Yaskawa INFORM job: R1_W14,16(0,0)OK-KM.JBI

/JOB
//NAME R1_W14,16(0,0)OK-KM
///FOLDERNAME KRIS-SCIANA
//POS
///NPOS 101,101,0,6,0,0
///TOOL 0
///POSTYPE PULSE
///PULSE
C00000=77640,24989,-13034,1442,74650,-81979
C00001=222133,14236,-6582,35909,75412,-22741
C00002=224151,18213,-1142,35502,73514,-22529
C00003=224936,19873,1121,35352,72748,-22454
C00004=225158,22602,3700,35316,72503,-22444
C00005=224936,19873,1121,35352,72748,-22454
C00006=225492,20065,2012,35260,72151,-22417
C00007=225492,20150,3698,35437,71333,-22690
C00008=225492,20065,2012,35260,72151,-22417
C00009=225905,19824,2070,35161,71851,-22342
C00010=226863,19321,1598,34859,71490,-22055
C00011=225905,19824,2070,35161,71851,-22342
C00012=225128,18122,-233,35305,72616,-22417
C00013=223128,14040,-5766,35700,74509,-22627
C00014=220661,2218,-15559,48375,67876,-23710
C00015=223949,9044,-9659,47271,66070,-22948
C00016=224087,10523,-8349,47237,65966,-22927
C00017=224042,10033,-8784,47248,66001,-22933
C00018=224042,10033,-8784,47248,66001,-22933
C00019=224745,9640,-9133,46989,65646,-22751
C00020=223995,9217,-9507,47256,66043,-22935
C00021=219810,-7663,-21002,65356,59757,-26400
C00022=222255,-3125,-17635,64445,58296,-25854
C00023=223197,-1261,-16218,64086,57730,-25645
C00024=223480,1501,-13911,63991,57548,-25594
C00025=223197,-1261,-16218,64086,57730,-25645
C00026=223908,-1254,-16349,63799,57315,-25476
C00027=225105,-1875,-16864,63387,56549,-25256
C00028=223908,-1254,-16349,63799,57315,-25476
C00029=223463,-1317,-18857,63116,58306,-24835
C00030=223463,-1302,-19472,62908,58490,-24651
C00031=223424,-1704,-17925,63552,57967,-25210
C00032=222481,-3577,-19346,63923,58526,-25421
C00033=220036,-8144,-22725,64866,59971,-25975
C00034=226102,-30423,-43926,14586,59978,3306
C00035=229259,38452,3699,-28321,84051,11178
C00036=227866,42540,10325,-28019,81848,11201
C00037=226976,47240,16142,-27837,80525,11190
C00038=226976,47162,16651,-27859,80211,11267
C00039=226976,47240,16142,-27837,80525,11190
C00040=223490,38048,5548,-21341,76491,4888
C00041=223597,39362,6909,-21393,76366,4949
C00042=225154,40482,8624,-23914,78071,7653
C00043=226382,33405,5149,-28983,73314,10641
C00044=225848,33713,5458,-28793,73102,10489
C00045=226800,33173,4915,-29132,73476,10760
C00046=227343,31188,2133,-29239,74267,10763
C00047=228749,26406,-4564,-29549,76202,10795
C00048=232070,-21849,-33765,-61090,62787,20907
C00049=228897,-69525,-52932,-81421,40129,27644
C00050=227458,-1039,11305,-103194,37608,33319
C00051=224958,9874,17770,-101661,35535,32336
C00052=224188,13683,20614,-101562,34950,32247
C00053=224309,15055,21867,-101627,35049,32289
C00054=224188,13683,20614,-101562,34950,32247
C00055=228943,22603,28948,-98890,46973,31456
C00056=228371,22871,29203,-99004,46566,31500
C00057=230119,20169,17224,-83081,48510,27787
C00058=230119,19939,16315,-82693,48579,27522
C00059=230119,20412,18152,-83475,48444,28057
C00060=230834,18316,16575,-83629,48946,28167
C00061=237272,-16480,-7416,-86396,53244,30318
C00062=226102,-30423,-43926,14586,59978,18513
C00063=216741,-24945,-44490,70900,55443,-67548
C00064=233770,-38242,-44235,89025,19285,-70455
C00065=232263,-12981,-20271,101799,31607,-56551
C00066=225008,-3810,-25351,68302,49674,-66777
C00067=224928,-2342,-24150,68324,49732,-66782
C00068=232472,-143,20091,126873,38436,-70149
C00069=232295,-11422,-4289,83587,31547,-48271
C00070=235949,-23068,-3497,134153,23753,-86044
C00071=221775,-4145,-3632,80714,47909,-75071
C00072=221868,-5805,-11746,98440,47173,-76002
C00073=224762,-3456,-10718,97920,45016,-75779
C00074=212311,-14192,-18848,96672,72508,-34975
C00075=225062,-3438,-11050,97706,44778,-75655
C00076=224981,-1976,-9851,97692,44835,-75643
C00077=212303,2769,29618,102443,75165,-45073
C00078=223552,-52882,-25947,90849,39544,-36058
C00079=221750,-4780,-5976,79726,48150,-74402
C00080=222455,-35947,-31649,13557,42914,-27667
C00081=237520,-26297,-36521,-56184,44849,52997
C00082=227430,-8986,2777,-105996,27008,67297
C00083=226046,668,8189,-102778,26699,65688
C00084=225096,7310,14013,-103452,26054,65991
C00085=227562,6691,-16510,-46000,42357,47609
C00086=227319,5585,-17469,-45803,42251,47516
C00087=224970,42335,84441,-140073,39060,85063
C00088=224879,29476,62062,-121250,29359,73886
C00089=227160,29335,71248,-136736,39012,83614
C00090=229934,2939,2236,-61070,35416,56138
C00091=229942,357,-16619,-50330,41431,49996
C00092=230607,-744,-7505,-83554,33312,60975
C00093=228290,3572,-4729,-82188,31724,60324
C00094=227452,5680,-3434,-81484,31174,59986
C00095=228279,4951,-3893,-81869,31750,60157
C00096=228037,3832,-4852,-81778,31579,60118
C00097=227208,23451,46622,-116903,33779,78542
C00098=230396,11237,36356,-114852,35808,77806
C00099=237476,-68885,-64231,-58705,66532,55214
C00100=145215,-69093,-87212,-37312,66696,68321
BC00000=241198,366988,1031591
BC00001=398174,77442,788239
BC00002=398174,77442,788239
BC00003=398174,77442,788239
BC00004=398174,77442,788239
BC00005=398174,77442,788239
BC00006=398174,77442,788239
BC00007=398174,77442,788239
BC00008=398174,77442,788239
BC00009=398174,77442,788239
BC00010=398174,77442,788239
BC00011=398174,77442,788239
BC00012=398174,77442,788239
BC00013=398174,77442,788239
BC00014=398174,70944,901946
BC00015=398174,70944,901946
BC00016=398174,70944,901946
BC00017=398174,70944,901946
BC00018=398174,70944,901946
BC00019=398174,70944,901946
BC00020=398174,70944,901946
BC00021=398174,63251,1036573
BC00022=398174,63251,1036573
BC00023=398174,63251,1036573
BC00024=398174,63251,1036573
BC00025=398174,63251,1036573
BC00026=398174,63251,1036573
BC00027=398174,63251,1036573
BC00028=398174,63251,1036573
BC00029=398174,63251,1036573
BC00030=398174,63251,1036573
BC00031=398174,63251,1036573
BC00032=398174,63251,1036573
BC00033=398174,63251,1036573
BC00034=398174,59868,1073520
BC00035=398174,86212,734350
BC00036=398174,86212,734350
BC00037=398174,86212,734350
BC00038=398174,86212,734350
BC00039=398174,86212,734350
BC00040=398174,86212,734350
BC00041=398174,86212,734350
BC00042=398174,86212,734350
BC00043=398174,86212,734350
BC00044=398174,86212,734350
BC00045=398174,86212,734350
BC00046=398174,86212,734350
BC00047=398174,86212,734350
BC00048=398174,98499,866647
BC00049=398174,100680,959819
BC00050=398174,103382,1075175
BC00051=398174,103382,1075175
BC00052=398174,103382,1075175
BC00053=398174,103382,1075175
BC00054=398174,103382,1075175
BC00055=398174,103382,1075175
BC00056=398174,103382,1075175
BC00057=398174,103382,1075175
BC00058=398174,103382,1075175
BC00059=398174,103382,1075175
BC00060=398174,103382,1075175
BC00061=398174,103382,1075175
BC00062=395324,71612,1073520
BC00063=398174,59556,681470
BC00064=398173,59556,681467
BC00065=398172,59557,681466
BC00066=398174,59556,681470
BC00067=398174,59556,681470
BC00068=398172,59557,681466
BC00069=398172,59557,681466
BC00070=398173,59556,681467
BC00071=398174,59556,681470
BC00072=398174,59378,943465
BC00073=398174,59378,943465
BC00074=355798,67513,940049
BC00075=398174,59378,943465
BC00076=398174,59378,943465
BC00077=355868,67500,939621
BC00078=355790,67515,940051
BC00079=398174,59378,943465
BC00080=398174,70552,906013
BC00081=398174,90929,866532
BC00082=398173,90931,866530
BC00083=398173,90931,866530
BC00084=398173,90931,866530
BC00085=398174,90929,866532
BC00086=398174,90929,866532
BC00087=398173,90931,866530
BC00088=398173,90931,866530
BC00089=398173,90931,866530
BC00090=398174,90929,866532
BC00091=398174,90929,866532
BC00092=398174,91899,990889
BC00093=398174,91899,990889
BC00094=398174,91900,990886
BC00095=398174,91899,990889
BC00096=398174,91899,990889
BC00097=398174,91899,990889
BC00098=398174,91899,990889
BC00099=398174,91899,990889
BC00100=363350,486581,1028471
///POSTYPE BASE
///RECTAN
///RCONF 0,0,0,0,1,0,0,0,0,0,0,0,0,0,0,0,0,0,0,0,0,0,0,0
P00006=2.006,1.622,-0.565,0.0000,0.0000,0.0000
P00021=0.073,2.058,-0.109,0.0000,0.0000,0.0000
P00022=2.006,1.622,-0.565,0.0000,0.0000,0.0000
///RCONF 0,0,0,0,0,0,0,0,0,0,0,0,0,0,0,0,0,0,0,0,0,0,0,0
P00023=-2.957,-4.083,2.762,0.0000,0.0000,0.0000
P00024=-1.466,-0.226,-0.419,0.0000,0.0000,0.0000
P00025=3.643,0.007,-2.585,0.0000,0.0000,0.0000
//INST
///DATE 2025/04/11 11:13
///ATTR SC,RW
///GROUP1 RB1,BS1
NOP
'r1_W14,16(0,0)
'Path S915
SFTOF
MOVJ C00000 BC00000 VJ=100.00
MOVL C00001 BC00001 V=333.3
MOVL C00002 BC00002 V=250.0
MOVL C00003 BC00003 V=60.0
REFP 3 C00004 BC00004
CALL JOB:SEARCH-R1
SET P021 P006
SFTON P021
MOVL C00005 BC00005 V=60.0
MOVL C00006 BC00006 V=60.0
REFP 3 C00007 BC00007
CALL JOB:SEARCH-R1
SET P021 P006
SFTON P021
MOVL C00008 BC00008 V=60.0
MOVL C00009 BC00009 V=60.0
REFP 3 C00010 BC00010
CALL JOB:SEARCH-R1
SET P021 P006
SFTON P021
MOVL C00011 BC00011 V=60.0
MOVL C00012 BC00012 V=166.7
MOVL C00013 BC00013 V=166.7
'Path S795 (for W413)
SFTOF
MOVL C00014 BC00014 V=166.7
MOVL C00015 BC00015 V=60.0
REFP 3 C00016 BC00016
CALL JOB:SEARCH-R1
SET P025 P006
SFTON P025
MOVL C00017 BC00017 V=60.0
MOVL C00018 BC00018 V=60.0
REFP 3 C00019 BC00019
CALL JOB:SEARCH-R1
SET P025 P006
SFTON P025
MOVL C00020 BC00020 V=60.0
MOVL C00021 BC00021 V=166.7
MOVL C00022 BC00022 V=166.7
MOVL C00023 BC00023 V=60.0
REFP 3 C00024 BC00024
CALL JOB:SEARCH-R1
SET P022 P006
SFTON P022
MOVL C00025 BC00025 V=60.0
MOVL C00026 BC00026 V=60.0
REFP 3 C00027 BC00027
CALL JOB:SEARCH-R1
SET P022 P006
SFTON P022
MOVL C00028 BC00028 V=60.0
MOVL C00029 BC00029 V=60.0
REFP 3 C00030 BC00030
CALL JOB:SEARCH-R1
SET P022 P006
SFTON P022
MOVL C00031 BC00031 V=166.7
MOVL C00032 BC00032 V=166.7
MOVL C00033 BC00033 V=166.7
MOVJ C00034 BC00034 VJ=100.00
'Path S806 (for W414)
SFTOF
MOVL C00035 BC00035 V=333.3
MOVL C00036 BC00036 V=250.0
MOVL C00037 BC00037 V=60.0
REFP 3 C00038 BC00038
CALL JOB:SEARCH-R1
SET P023 P006
SFTON P023
MOVL C00039 BC00039 V=60.0
MOVL C00040 BC00040 V=60.0
REFP 3 C00041 BC00041
CALL JOB:SEARCH-R1
SET P023 P006
SFTON P023
MOVL C00042 BC00042 V=60.0
MOVL C00043 BC00043 V=60.0
REFP 3 C00044 BC00044
CALL JOB:SEARCH-R1
SET P023 P006
SFTON P023
MOVL C00045 BC00045 V=60.0
MOVL C00046 BC00046 V=166.7
MOVL C00047 BC00047 V=166.7
MOVJ C00048 BC00048 VJ=100.00
'Path VIA1130
SFTOF
MOVJ C00049 BC00049 VJ=100.00
'Path S807 (for W414)
SFTOF
MOVJ C00050 BC00050 VJ=100.00
MOVJ C00051 BC00051 VJ=100.00
MOVL C00052 BC00052 V=60.0
REFP 3 C00053 BC00053
CALL JOB:SEARCH-R1
SET P024 P006
SFTON P024
MOVL C00054 BC00054 V=60.0
MOVL C00055 BC00055 V=60.0
REFP 3 C00056 BC00056
CALL JOB:SEARCH-R1
SET P024 P006
SFTON P024
MOVL C00057 BC00057 V=60.0
REFP 3 C00058 BC00058
CALL JOB:SEARCH-R1
SET P024 P006
SFTON P024
MOVL C00059 BC00059 V=116.7
MOVL C00060 BC00060 V=333.3
MOVL C00061 BC00061 V=333.3
MOVJ C00062 BC00062 VJ=100.00
'Path W1128
SFTOF
CALL JOB:COFNIJ_DRUT
SFTON P025
MOVJ C00063 BC00063 VJ=100.00
MOVJ C00064 BC00064 VJ=100.00
MOVL C00065 BC00065 V=100.0 PL=0
REFP 1 C00066 BC00066
REFP 2 C00067 BC00067
MACRO1 MJ#(0) ARGF7
ARCON
SFTON P021
MOVL C00068 BC00068 V=14.2
MOVL C00069 BC00069 V=14.2
ARCOF
MOVL C00070 BC00070 V=166.7
MOVL C00071 BC00071 V=166.7
SFTOF
'Path W1129
SFTOF
SFTON P022
MOVJ C00072 BC00072 VJ=100.00
MOVJ C00073 BC00073 VJ=100.00
MOVL C00074 BC00074 V=166.7 PL=0
REFP 1 C00075 BC00075
REFP 2 C00076 BC00076
MACRO1 MJ#(0) ARGF7
ARCON
SFTON P025
MOVL C00077 BC00077 V=14.2 PL=0
ARCOF
MOVL C00078 BC00078 V=166.7
MOVL C00079 BC00079 V=166.7
SFTOF
'Path VIA1131
SFTOF
MOVJ C00080 BC00080 VJ=100.00
'Path W868
SFTOF
SFTON P024
MOVJ C00081 BC00081 VJ=100.00
MOVJ C00082 BC00082 VJ=45.00
MOVJ C00083 BC00083 VJ=100.00
MOVL C00084 BC00084 V=100.0 PL=0
REFP 1 C00085 BC00085
REFP 2 C00086 BC00086
MACRO1 MJ#(0) ARGF10
ARCON
SFTON P023
MOVL C00087 BC00087 V=10.0
MOVL C00088 BC00088 V=10.0
ARCOF
MOVL C00089 BC00089 V=166.7
MOVL C00090 BC00090 V=166.7
MOVL C00091 BC00091 V=166.7
SFTOF
'Path W1127
SFTOF
'Path W1126
SFTOF
SFTON P024
MOVJ C00092 BC00092 VJ=100.00
MOVJ C00093 BC00093 VJ=100.00
MOVL C00094 BC00094 V=100.0 PL=0
REFP 1 C00095 BC00095
REFP 2 C00096 BC00096
MACRO1 MJ#(0) ARGF10
ARCON
SFTON P023
MOVL C00097 BC00097 V=10.0
ARCOF
MOVL C00098 BC00098 V=166.7
MOVL C00099 BC00099 V=333.3
MOVJ C00100 BC00100 VJ=100.00
SFTOF
END
